Staubli VAL3: Rectangle10.pjx

Parameters version=s7.7.1 stackSize=5000 millimeterUnit=true
Program file=start.pgx
Program file=stop.pgx
Data file=Rectangle10.dtx
